{attribute 'linkalways'} 
{attribute 'no_explicit_call' := 'This FB is a CLASS and must be accessed using methods or properties'}
{attribute 'enable_dynamic_creation'}
FUNCTION_BLOCK ExtensionHost IMPLEMENTS I_Extensions, I_Serializable, I_Deserializable
VAR
	hostParent : I_HostExtensions;
	eventTarget : I_EventTarget;
	extensions : Dictionary;
END_VAR

METHOD PUBLIC Accept
VAR_INPUT
	Visitor : I_ExtensionVisitor;
END_VAR
VAR
	enumerator : I_ForwardEnumerator;
	extension : I_Extension;
END_VAR
enumerator := extensions.GetEnumerator();

WHILE (enumerator.MoveNext()) DO
	
	IF enumerator.TryGet(extension) THEN
		extension.Accept(Visitor);
	END_IF

END_WHILE

enumerator.Dispose();
END_METHOD

METHOD PUBLIC AddExtension
VAR_INPUT
	Extension : I_Extension;
END_VAR
extensions.AddOrUpdate(Extension.Name,Extension);
EmitOnExtensionAddedEvent(Extension);
END_METHOD

METHOD PROTECTED EmitOnExtensionAddedEvent
VAR_INPUT
	Extension : I_Extension;
END_VAR
VAR
	pExtensionAddedEvent : POINTER TO ExtensionAddedEvent;
END_VAR
IF eventTarget = 0 THEN
	RETURN;
END_IF

pExtensionAddedEvent := __NEW(ExtensionAddedEvent(Target := Extension));
eventTarget.Emit('OnExtensionAdded',pExtensionAddedEvent^);
pExtensionAddedEvent^.Dispose();
END_METHOD

METHOD FB_init : BOOL
VAR_INPUT
	bInitRetains : BOOL; // if TRUE, the retain variables are initialized (warm start / cold start)
	bInCopyCode : BOOL;  // if TRUE, the instance afterwards gets moved into the copy code (online change)
	Parent : I_HostExtensions;
	ParentEventTarget : I_EventTarget;
END_VAR
hostParent := Parent;
eventTarget := parentEventTarget;
END_METHOD

PROPERTY PUBLIC HasExtensions : BOOL
GET
HasExtensions := extensions.Count > 0;
END_GET
END_PROPERTY

METHOD PUBLIC SerializeWith
VAR_INPUT
	Serializer : I_Serializer;
END_VAR
VAR
	enumerator : I_ForwardEnumerator;
	extension : I_Extension;
END_VAR
IF extensions.Count = 0 THEN
	RETURN;
END_IF

Serializer.AddKey('extensions');
Serializer.StartArray();

enumerator := extensions.GetEnumerator();

WHILE enumerator.MoveNext() DO
	IF enumerator.TryGet(extension) THEN
		extension.SerializeWith(Serializer);
	END_IF
END_WHILE

Serializer.EndArray();
enumerator.Dispose();
END_METHOD

METHOD public TryDeserializeFrom : BOOL
VAR_INPUT
	Deserializer : I_Deserializer;
	Feedback : I_DeserializerFeedback;
END_VAR
VAR
	extensionsDeserializer : I_Deserializer;
	extensionsEnumerator : I_DeserializerArrayForwardEnumerator;
	extensionName : T_MAXSTRING;
	extension : I_Extension;
END_VAR
extensionsDeserializer := Deserializer.GetKeyArray('extensions');
extensionsEnumerator := extensionsDeserializer.GetArrayEnumerator();

WHILE extensionsEnumerator.MoveNext() DO
	
	IF NOT extensionsEnumerator.Current.TryGetKeyString('name', extensionName, Feedback) THEN
		CONTINUE;
	END_IF
	
	IF NOT TryGetExtensionByName(extensionName, extension) THEN
		CONTINUE;
	END_IF
	
	IF NOT extension.TryDeserializeFrom(extensionsEnumerator.Current, Feedback) THEN
		extensionsEnumerator.Dispose();
		RETURN;
	END_IF

END_WHILE

TryDeserializeFrom := TRUE;
extensionsEnumerator.Dispose();
END_METHOD

METHOD PUBLIC TryGetExtensionByName : BOOL
VAR_INPUT
	Name : T_MAXSTRING;
	Destination : REFERENCE TO I_Extension;
END_VAR
VAR
	extension : I_Extension;
END_VAR
IF NOT extensions.TryGetValue(Name, extension) THEN
	RETURN;
END_IF

Destination := extension;
TryGetExtensionByName := TRUE;
END_METHOD

END_FUNCTION_BLOCK

(* stored: Version 1.1.0.1, ProductVersion 3.1.4024.12
   POU ExtensionHost: Id {1342cd0e-30df-4c6d-859e-45f9ea8ed804}, SpecialFunc None
   Folder Constructor: Id {0b596dd9-3dea-4016-8869-9183452b6fbd}
   Folder Protected: Id {428df022-7761-4cc4-8f9a-a96aace27d7a}
   Method Accept: Id {b9b3366b-2395-4b36-a0d4-c803ea45cfd2}
   Method AddExtension: Id {42b7879a-6c0b-409a-a931-045c18793742}
   Method EmitOnExtensionAddedEvent: Id {3db98306-6f82-4266-b66b-198643853dbe}
   Method FB_init: Id {4d716ee7-2d1a-4785-9f33-1378b60a0ebf}
   Property HasExtensions: Id {0d166c03-b0e6-0f93-1bdc-cbe61996891b}
   Get Get: Id {b88cc1f5-60c3-08df-2ef4-cbbcf44048c5}
   Method SerializeWith: Id {7cb20ebb-fbc3-4bf7-be48-3cce675f08ac}
   Method TryDeserializeFrom: Id {554559c6-e903-4586-95d7-5e80ef0e38a4}
   Method TryGetExtensionByName: Id {b998adb0-f111-4cb3-bea7-519b22b71849} *)
